Universal Robots PolyScope program: Grab_spoon.urp

Program Grab_spoon (installation=default directory=/programs/Matcha createdIn=5.12.6.1102099 lastSavedIn=5.12.6.1102099 robotSerialNumber=20215500597)
Calibrated DH parameters: a=[0.000193, -0.066673, -0.391568, -0.000012, 0.00005, 0]; d=[0.162643, -472.05677, 465.132521, 7.058239, 0.099746, 0.099582]; alpha=[1.571116, 0.00089, 0.003862, 1.569269, -1.569248, 0]; deltaTheta=[0, -1.413394, 7.628392, 0.068187, 0, -0.000001]
Robot Program (runOnlyOnce=true)
  MoveJ speed 60 deg/s, acceleration 80 deg/s^2 (useActiveTCP=true) feature=Base
    Waypoint spoonhome: TCP in base x=-57.019 y=-490.097 z=96.977 mm, rx=-0.014 ry=1.5917 rz=-0.0244 rad; joints [41.639, -46.218, 88.996, -44.212, -47.879, -90.492] deg; TCP offset x=0 y=0 z=191.5 mm, rx=0 ry=0 rz=0 rad
  URCap Gripper Activate (Robotiq_Grippers, Robotiq Inc.) dataModel(ResetAndActivateKey=false)
  URCap Gripper (Robotiq_Grippers, Robotiq Inc.) dataModel(position=59.2156862745098, force=0.0, speed=0.0, positionInDouble=59.2156862745098, forceInDouble=0.0, speedInDouble=0.0, slaveIds=[9], blocking=true)
  spoon := GP_int_in[0]
  y_offset := p[0,-0.055*spoon,0,0,0,0]
  x_offset := p[0.17964,0,0,0,0,0]
  z_offset := p[0,0,0.04762,0,0,0]
  spoon_pos := pose_add(matchaSpoonHome, y_offset)
  grab_back_pos := pose_add(spoon_pos, x_offset)
  grab_hover_pose := pose_add(grab_back_pos, z_offset)
  MoveL speed 250 mm/s, acceleration 1200 mm/s^2 (useActiveTCP=true) feature=Base
    Waypoint Waypoint (Variable): variable=matchaSpoonHome
    Waypoint Waypoint (Variable): variable=spoon_pos
    Waypoint Waypoint (Variable): variable=grab_back_pos
    URCap Gripper (Robotiq_Grippers, Robotiq Inc.) dataModel(position=88.88235294117646, force=0.0, speed=0.0, positionInDouble=88.88235294117646, forceInDouble=0.0, speedInDouble=0.0, slaveIds=[9], blocking=true)
    Waypoint Waypoint (Variable): variable=grab_hover_pose
    Waypoint Waypoint (Variable): variable=spoon_pos
    Waypoint spoonhome: TCP in base x=-57.019 y=-490.097 z=96.977 mm, rx=-0.014 ry=1.5917 rz=-0.0244 rad; joints [41.639, -46.218, 88.996, -44.212, -47.879, -90.492] deg
